FUNCTION_BLOCK PROCESS_SC (* Peroidic event generator *)
  (* Standard: 61499-1 Annex A; Description: Copyright (c) 2017 fortiss GmbH This program and the accompanying materials are made available under the terms of the Eclipse Public License 2.0 which is available at https://www.eclipse.org/legal/epl-2.0/ SPDX-License-Identifier: EPL-2.0 *)
  (* Version 1.0, 2017-09-21, Alois Zoitl, fortiss GmbH, initial API and implementation and/or initial documentation *)
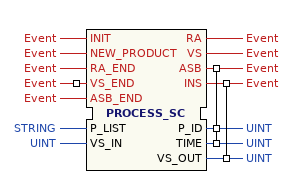
  EVENT_INPUT
    INIT;
    NEW_PRODUCT;
    RA_END;
    VS_END WITH VS_OUT;
    ASB_END;
  END_EVENT
  EVENT_OUTPUT
    RA;
    VS;
    ASB WITH P_ID, TIME;
    INS WITH VS_OUT;
  END_EVENT
  VAR_INPUT
    P_LIST : STRING;
    VS_IN : UINT;
  END_VAR
  VAR_OUTPUT
    P_ID : UINT;
    TIME : UINT;
    VS_OUT : UINT;
  END_VAR
END_FUNCTION_BLOCK
